// TIA Portal V20 export
FUNCTION_BLOCK "LER_StackTableVisionConversion"   // FB125, LAD
// stored: Access Published, MemoryReserve 100, SetENOAutomatically false
   VAR_INPUT
      VisionData : "LER_typeVisionMonitoring";
   END_VAR
   VAR_OUTPUT
      VisionDataConvert : "LER_typeVisionGapResultData";
   END_VAR
BEGIN

REGION Network 1 (SCL)
   // Result
   #VisionDataConvert.visionLengthOfSeparatorCathodeJudgementResult := 0.001 * DINT_TO_REAL(#VisionData.profinetInput.resultData248Byte_1.resultData[0]);
   #VisionDataConvert.visionLengthOfSeparatorAnodeJudgementResult   := 0.001 * DINT_TO_REAL(#VisionData.profinetInput.resultData248Byte_1.resultData[1]);
   #VisionDataConvert.visionCathodeLengthJudgementResult := 0.001 * DINT_TO_REAL(#VisionData.profinetInput.resultData248Byte_1.resultData[2]);
   #VisionDataConvert.visionAnodeLengthJudgementResult := 0.001 * DINT_TO_REAL(#VisionData.profinetInput.resultData248Byte_1.resultData[3]);
   #VisionDataConvert.visionCathodeToSeparatorY1JudgementResult := 0.001 * DINT_TO_REAL(#VisionData.profinetInput.resultData248Byte_1.resultData[4]);
   #VisionDataConvert.visionCathodeToSeparatorY2JudgementResult := 0.001 * DINT_TO_REAL(#VisionData.profinetInput.resultData248Byte_1.resultData[5]);
   #VisionDataConvert.visionCathodeToSeparatorY3JudgementResult := 0.001 * DINT_TO_REAL(#VisionData.profinetInput.resultData248Byte_1.resultData[6]);
   #VisionDataConvert.visionCathodeToSeparatorY4JudgementResult := 0.001 * DINT_TO_REAL(#VisionData.profinetInput.resultData248Byte_1.resultData[7]);
   #VisionDataConvert.visionCathodeToAnodeY1JudgementResult := 0.001 * DINT_TO_REAL(#VisionData.profinetInput.resultData248Byte_1.resultData[8]);
   #VisionDataConvert.visionCathodeToAnodeY2JudgementResult := 0.001 * DINT_TO_REAL(#VisionData.profinetInput.resultData248Byte_1.resultData[9]);
   #VisionDataConvert.visionAnodeToCathodeY1JudgementResult := 0.001 * DINT_TO_REAL(#VisionData.profinetInput.resultData248Byte_1.resultData[10]);
   #VisionDataConvert.visionAnodeToCathodeY2JudgementResult := 0.001 * DINT_TO_REAL(#VisionData.profinetInput.resultData248Byte_1.resultData[11]);
   #VisionDataConvert.visionAnodeToSeparatorY1JudgementResult := 0.001 * DINT_TO_REAL(#VisionData.profinetInput.resultData248Byte_1.resultData[12]);
   #VisionDataConvert.visionAnodeToSeparatorY2JudgementResult := 0.001 * DINT_TO_REAL(#VisionData.profinetInput.resultData248Byte_1.resultData[13]);
   #VisionDataConvert.visionAnodeToCathodeX1JudgementResult := 0.001 * DINT_TO_REAL(#VisionData.profinetInput.resultData248Byte_1.resultData[14]);
   #VisionDataConvert.visionAnodeToCathodeX2JudgementResult := 0.001 * DINT_TO_REAL(#VisionData.profinetInput.resultData248Byte_1.resultData[15]);
   #VisionDataConvert.visionAnodeToCathodeX3JudgementResult := 0.001 * DINT_TO_REAL(#VisionData.profinetInput.resultData248Byte_1.resultData[16]);
   #VisionDataConvert.visionAnodeToCathodeX4JudgementResult := 0.001 * DINT_TO_REAL(#VisionData.profinetInput.resultData248Byte_1.resultData[17]);
   #VisionDataConvert.visionCathodeToSeparatorX1JudgementResult := 0.001 * DINT_TO_REAL(#VisionData.profinetInput.resultData248Byte_1.resultData[18]);
   #VisionDataConvert.visionCathodeToSeparatorX2JudgementResult := 0.001 * DINT_TO_REAL(#VisionData.profinetInput.resultData248Byte_1.resultData[19]);
   #VisionDataConvert.visionCathodeToSeparatorX3JudgementResult := 0.001 * DINT_TO_REAL(#VisionData.profinetInput.resultData248Byte_1.resultData[20]);
   #VisionDataConvert.visionCathodeToSeparatorX4JudgementResult := 0.001 * DINT_TO_REAL(#VisionData.profinetInput.resultData248Byte_1.resultData[21]);
   #VisionDataConvert.visionAnodeToSeparatorX1JudgementResult := 0.001 * DINT_TO_REAL(#VisionData.profinetInput.resultData248Byte_1.resultData[22]);
   #VisionDataConvert.visionAnodeToSeparatorX2JudgementResult := 0.001 * DINT_TO_REAL(#VisionData.profinetInput.resultData248Byte_1.resultData[23]);
   #VisionDataConvert.visionAnodeToSeparatorX3JudgementResult := 0.001 * DINT_TO_REAL(#VisionData.profinetInput.resultData248Byte_1.resultData[24]);
   #VisionDataConvert.visionAnodeToSeparatorX4JudgementResult := 0.001 * DINT_TO_REAL(#VisionData.profinetInput.resultData248Byte_1.resultData[25]);

   // Measured value
   #VisionDataConvert.visionLengthOfSeparatorCathodeReply := DINT_TO_REAL(#VisionData.profinetInput.resultData248Byte_1.resultData[26]);
   #VisionDataConvert.visionLengthOfSeparatorCathodeUpperRangeReply := DINT_TO_REAL(#VisionData.profinetInput.resultData248Byte_1.resultData[27]);
   #VisionDataConvert.visionLengthOfSeparatorCathodeLowerRangeReply := DINT_TO_REAL(#VisionData.profinetInput.resultData248Byte_1.resultData[28]);
   #VisionDataConvert.visionLengthOfSeparatorAnodeReply := DINT_TO_REAL(#VisionData.profinetInput.resultData248Byte_1.resultData[29]);
   #VisionDataConvert.visionLengthOfSeparatorAnodeUpperRangeReply := DINT_TO_REAL(#VisionData.profinetInput.resultData248Byte_1.resultData[30]);
   #VisionDataConvert.visionLengthOfSeparatorAnodeLowerRangeReply := DINT_TO_REAL(#VisionData.profinetInput.resultData248Byte_1.resultData[31]);
   #VisionDataConvert.visionCathodeLengthReply := DINT_TO_REAL(#VisionData.profinetInput.resultData248Byte_1.resultData[32]);
   #VisionDataConvert.visionCathodeLengthUpperRangeReply := DINT_TO_REAL(#VisionData.profinetInput.resultData248Byte_1.resultData[33]);
   #VisionDataConvert.visionCathodeLengthLowerRangeReply := DINT_TO_REAL(#VisionData.profinetInput.resultData248Byte_2[0]);
   #VisionDataConvert.visionAnodeLengthReply := DINT_TO_REAL(#VisionData.profinetInput.resultData248Byte_2[1]);
   #VisionDataConvert.visionAnodeLengthUpperRangeReply := DINT_TO_REAL(#VisionData.profinetInput.resultData248Byte_2[2]);
   #VisionDataConvert.visionAnodeLengthLowerRangeReply := DINT_TO_REAL(#VisionData.profinetInput.resultData248Byte_2[3]);
   #VisionDataConvert.visionCathodeToSeparatorY1Reply := DINT_TO_REAL(#VisionData.profinetInput.resultData248Byte_2[4]);
   #VisionDataConvert.visionCathodeToSeparatorY1UpperRangeReply := DINT_TO_REAL(#VisionData.profinetInput.resultData248Byte_2[5]);
   #VisionDataConvert.visionCathodeToSeparatorY1LowerRangeReply := DINT_TO_REAL(#VisionData.profinetInput.resultData248Byte_2[6]);
   #VisionDataConvert.visionCathodeToSeparatorY2Reply := DINT_TO_REAL(#VisionData.profinetInput.resultData248Byte_2[7]);
   #VisionDataConvert.visionCathodeToSeparatorY2UpperRangeReply := DINT_TO_REAL(#VisionData.profinetInput.resultData248Byte_2[8]);
   #VisionDataConvert.visionCathodeToSeparatorY2LowerRangeReply := DINT_TO_REAL(#VisionData.profinetInput.resultData248Byte_2[9]);
   #VisionDataConvert.visionCathodeToSeparatorY3Reply := DINT_TO_REAL(#VisionData.profinetInput.resultData248Byte_2[10]);
   #VisionDataConvert.visionCathodeToSeparatorY3UpperRangeReply := DINT_TO_REAL(#VisionData.profinetInput.resultData248Byte_2[11]);
   #VisionDataConvert.visionCathodeToSeparatorY3LowerRangeReply := DINT_TO_REAL(#VisionData.profinetInput.resultData248Byte_2[12]);
   #VisionDataConvert.visionCathodeToSeparatorY4Reply := DINT_TO_REAL(#VisionData.profinetInput.resultData248Byte_2[13]);
   #VisionDataConvert.visionCathodeToSeparatorY4UpperRangeReply := DINT_TO_REAL(#VisionData.profinetInput.resultData248Byte_2[14]);
   #VisionDataConvert.visionCathodeToSeparatorY4LowerRangeReply := DINT_TO_REAL(#VisionData.profinetInput.resultData248Byte_2[15]);
   #VisionDataConvert.visionCathodeToAnodeY1Reply := DINT_TO_REAL(#VisionData.profinetInput.resultData248Byte_2[16]);
   #VisionDataConvert.visionCathodeToAnodeY1UpperRangeReply := DINT_TO_REAL(#VisionData.profinetInput.resultData248Byte_2[17]);
   #VisionDataConvert.visionCathodeToAnodeY1LowerRangeReply := DINT_TO_REAL(#VisionData.profinetInput.resultData248Byte_2[18]);
   #VisionDataConvert.visionCathodeToAnodeY2Reply := DINT_TO_REAL(#VisionData.profinetInput.resultData248Byte_2[19]);
   #VisionDataConvert.visionCathodeToAnodeY2UpperRangeReply := DINT_TO_REAL(#VisionData.profinetInput.resultData248Byte_2[20]);
   #VisionDataConvert.visionCathodeToAnodeY2LowerRangeReply := DINT_TO_REAL(#VisionData.profinetInput.resultData248Byte_2[21]);
   #VisionDataConvert.visionAnodeToCathodeY1Reply := DINT_TO_REAL(#VisionData.profinetInput.resultData248Byte_2[22]);
   #VisionDataConvert.visionAnodeToCathodeY1UpperRangeReply := DINT_TO_REAL(#VisionData.profinetInput.resultData248Byte_2[23]);
   #VisionDataConvert.visionAnodeToCathodeY1LowerRangeReply := DINT_TO_REAL(#VisionData.profinetInput.resultData248Byte_2[24]);
   #VisionDataConvert.visionAnodeToCathodeY2Reply := DINT_TO_REAL(#VisionData.profinetInput.resultData248Byte_2[25]);
   #VisionDataConvert.visionAnodeToCathodeY2UpperRangeReply := DINT_TO_REAL(#VisionData.profinetInput.resultData248Byte_2[26]);
   #VisionDataConvert.visionAnodeToCathodeY2LowerRangeReply := DINT_TO_REAL(#VisionData.profinetInput.resultData248Byte_2[27]);
   #VisionDataConvert.visionAnodeToSeparatorY1Reply := DINT_TO_REAL(#VisionData.profinetInput.resultData248Byte_2[28]);
   #VisionDataConvert.visionAnodeToSeparatorY1UpperRangeReply := DINT_TO_REAL(#VisionData.profinetInput.resultData248Byte_2[29]);
   #VisionDataConvert.visionAnodeToSeparatorY1LowerRangeReply := DINT_TO_REAL(#VisionData.profinetInput.resultData248Byte_2[30]);
   #VisionDataConvert.visionAnodeToSeparatorY2Reply := DINT_TO_REAL(#VisionData.profinetInput.resultData248Byte_2[31]);
   #VisionDataConvert.visionAnodeToSeparatorY2UpperRangeReply := DINT_TO_REAL(#VisionData.profinetInput.resultData248Byte_2[32]);
   #VisionDataConvert.visionAnodeToSeparatorY2LowerRangeReply := DINT_TO_REAL(#VisionData.profinetInput.resultData248Byte_2[33]);
   #VisionDataConvert.visionAnodeToCathodeX1Reply := DINT_TO_REAL(#VisionData.profinetInput.resultData248Byte_2[34]);
   #VisionDataConvert.visionAnodeToCathodeX1UpperRangeReply := DINT_TO_REAL(#VisionData.profinetInput.resultData248Byte_2[35]);
   #VisionDataConvert.visionAnodeToCathodeX1LowerRangeReply := DINT_TO_REAL(#VisionData.profinetInput.resultData248Byte_2[36]);
   #VisionDataConvert.visionAnodeToCathodeX2Reply := DINT_TO_REAL(#VisionData.profinetInput.resultData248Byte_2[37]);
   #VisionDataConvert.visionAnodeToCathodeX2UpperRangeReply := DINT_TO_REAL(#VisionData.profinetInput.resultData248Byte_2[38]);
   #VisionDataConvert.visionAnodeToCathodeX2LowerRangeReply := DINT_TO_REAL(#VisionData.profinetInput.resultData248Byte_2[39]);
   #VisionDataConvert.visionAnodeToCathodeX3Reply := DINT_TO_REAL(#VisionData.profinetInput.resultData248Byte_2[40]);
   #VisionDataConvert.visionAnodeToCathodeX3UpperRangeReply := DINT_TO_REAL(#VisionData.profinetInput.resultData248Byte_2[41]);
   #VisionDataConvert.visionAnodeToCathodeX3LowerRangeReply := DINT_TO_REAL(#VisionData.profinetInput.resultData248Byte_2[42]);
   #VisionDataConvert.visionAnodeToCathodeX4Reply := DINT_TO_REAL(#VisionData.profinetInput.resultData248Byte_2[43]);
   #VisionDataConvert.visionAnodeToCathodeX4UpperRangeReply := DINT_TO_REAL(#VisionData.profinetInput.resultData248Byte_2[44]);
   #VisionDataConvert.visionAnodeToCathodeX4LowerRangeReply := DINT_TO_REAL(#VisionData.profinetInput.resultData248Byte_2[45]);
   #VisionDataConvert.visionCathodeToSeparatorX1Reply := DINT_TO_REAL(#VisionData.profinetInput.resultData248Byte_2[46]);
   #VisionDataConvert.visionCathodeToSeparatorX1UpperRangeReply := DINT_TO_REAL(#VisionData.profinetInput.resultData248Byte_2[47]);
   #VisionDataConvert.visionCathodeToSeparatorX1LowerRangeReply := DINT_TO_REAL(#VisionData.profinetInput.resultData248Byte_2[48]);
   #VisionDataConvert.visionCathodeToSeparatorX2Reply := DINT_TO_REAL(#VisionData.profinetInput.resultData248Byte_2[49]);
   #VisionDataConvert.visionCathodeToSeparatorX2UpperRangeReply := DINT_TO_REAL(#VisionData.profinetInput.resultData248Byte_2[50]);
   #VisionDataConvert.visionCathodeToSeparatorX2LowerRangeReply := DINT_TO_REAL(#VisionData.profinetInput.resultData248Byte_2[51]);
   #VisionDataConvert.visionCathodeToSeparatorX3Reply := DINT_TO_REAL(#VisionData.profinetInput.resultData248Byte_2[52]);
   #VisionDataConvert.visionCathodeToSeparatorX3UpperRangeReply := DINT_TO_REAL(#VisionData.profinetInput.resultData248Byte_2[53]);
   #VisionDataConvert.visionCathodeToSeparatorX3LowerRangeReply := DINT_TO_REAL(#VisionData.profinetInput.resultData248Byte_2[54]);
   #VisionDataConvert.visionCathodeToSeparatorX4Reply := DINT_TO_REAL(#VisionData.profinetInput.resultData248Byte_2[55]);
   #VisionDataConvert.visionCathodeToSeparatorX4UpperRangeReply := DINT_TO_REAL(#VisionData.profinetInput.resultData248Byte_2[56]);
   #VisionDataConvert.visionCathodeToSeparatorX4LowerRangeReply := DINT_TO_REAL(#VisionData.profinetInput.resultData248Byte_2[57]);
   #VisionDataConvert.visionAnodeToSeparatorX1Reply := DINT_TO_REAL(#VisionData.profinetInput.resultData248Byte_2[58]);
   #VisionDataConvert.visionAnodeToSeparatorX1UpperRangeReply := DINT_TO_REAL(#VisionData.profinetInput.resultData248Byte_2[59]);
   #VisionDataConvert.visionAnodeToSeparatorX1LowerRangeReply := DINT_TO_REAL(#VisionData.profinetInput.resultData248Byte_2[60]);
   #VisionDataConvert.visionAnodeToSeparatorX2Reply := DINT_TO_REAL(#VisionData.profinetInput.resultData248Byte_2[61]);
   #VisionDataConvert.visionAnodeToSeparatorX2UpperRangeReply := DINT_TO_REAL(#VisionData.profinetInput.resultData248Byte_3[0]);
   #VisionDataConvert.visionAnodeToSeparatorX2LowerRangeReply := DINT_TO_REAL(#VisionData.profinetInput.resultData248Byte_3[1]);
   #VisionDataConvert.visionAnodeToSeparatorX3Reply := DINT_TO_REAL(#VisionData.profinetInput.resultData248Byte_3[2]);
   #VisionDataConvert.visionAnodeToSeparatorX3UpperRangeReply := DINT_TO_REAL(#VisionData.profinetInput.resultData248Byte_3[3]);
   #VisionDataConvert.visionAnodeToSeparatorX3LowerRangeReply := DINT_TO_REAL(#VisionData.profinetInput.resultData248Byte_3[4]);
   #VisionDataConvert.visionAnodeToSeparatorX4Reply := DINT_TO_REAL(#VisionData.profinetInput.resultData248Byte_3[5]);
   #VisionDataConvert.visionAnodeToSeparatorX4UpperRangeReply := DINT_TO_REAL(#VisionData.profinetInput.resultData248Byte_3[6]);
   #VisionDataConvert.visionAnodeToSeparatorX4LowerRangeReply := DINT_TO_REAL(#VisionData.profinetInput.resultData248Byte_3[7]);
END_REGION
END_FUNCTION_BLOCK
